FUNCTION_BLOCK FB_PrintModule_WEU_View
VAR
  // helper
  bInit   : BOOL;
  
  // config
  _pModule : POINTER TO FB_PrintModule_WEU;
  _pPositioning : POINTER TO FB_PrintPositionDmax;
  
  fbCTTrackerView : FB_CTTrackerView;
  
  // view selections
  nSelWorkerPrint : UDINT := 1;
  bShowFineAlignement : BOOL;
  // hardware view
  bShowPhDetail : BOOL;
  nSelPhDetail : UDINT := 1;
  bShowPcDetail : BOOL;
  nSelPcDetail : UDINT := 1;
  
  // motion and position view
  bShowPositionDetail : BOOL;
  bMovingInd : BOOL;
  fSpeed  : LREAL;
  fbBlink_Moving : FB_BLINK;
  
  // debug view
  bShowDebugAndSim : BOOL;
  
  fbBlink_Printing : FB_BLINK;
  bBlinkPrint : BOOL;
  bPrintInd : ARRAY[1..GVL_WEU.nC_MaxWorkerPrintPerPm] OF BOOL;
  fMaxPos : LREAL;
  t : TIME;
  zPos_PM : UDINT;
  i : UDINT;
END_VAR

VAR CONSTANT
  nC_MAX_WORKER_VIEWS : UINT := 10;
END_VAR

IF NOT checkConfig() THEN RETURN; END_IF    // check config

// -- show moving -----------------------
fSpeed := _pPositioning^.getSpeed();
IF LrealIsNaN(x:=fSpeed) THEN
  fSpeed := 0;
END_IF
t := LREAL_TO_TIME(1000-fSpeed*900);
fbBlink_Moving(bI_Enable:=SEL(fSpeed > 0, FALSE, TRUE), tI_Time:=t, bO_Out=>bMovingInd);

t := T#400MS;
fbBlink_Moving(bI_Enable:=TRUE, tI_Time:=t, bO_Out=>bBlinkPrint);
FOR i:=1 TO GVL_WEU.nC_MaxWorkerPrintPerPm DO
  bPrintInd[i] := _pModule^.fbWorkerPrint[i].bPrinting AND bBlinkPrint;
  fMaxPos := MAX(_pModule^.fbWorkerPrint[i].fPosition, fMaxPos);
END_FOR


// -- show pm module position
zPos_PM := SEL(_pModule^._pModuleMachineState^.bUnitInPrintPosition, 0, 40);

// -- show pg in p,
nSelWorkerPrint := LIMIT(1, nSelWorkerPrint, GVL_WEU.nC_MaxWorkerPrintPerPm);

// -- show ph detail
nSelPhDetail := LIMIT(1, nSelPhDetail, _pModule^._nPh);
nSelPcDetail := LIMIT(1, nSelPcDetail, _pModule^._nPc);

// -- CTTracker overview view
fbCTTrackerView.fX_m  := fMaxPos + 0.1;
fbCTTrackerView.fY_m  := 1;
fbCTTrackerView.nX_px := 300;
fbCTTrackerView.nY_px := 100;
fbCTTrackerView.fPxToMRatio := fbCTTrackerView.nX_px / fbCTTrackerView.fX_m;
fbCTTrackerView.iPrintPosition :=_pPositioning^;
fbCTTrackerView();

METHOD checkConfig : BOOL
VAR_INPUT
END_VAR
VAR_INST
  _fX_m, _fY_m   : LREAL;
  _nX_px, _nY_px : DINT; 
END_VAR
VAR
  bOK : BOOL;
END_VAR
IF NOT bInit THEN RETURN; END_IF

checkConfig := TRUE;
END_METHOD

METHOD init : BOOL
VAR_INPUT
  pModule : POINTER TO FB_PrintModule_WEU;
  pPositioning : POINTER TO FB_PrintPositionDmax;
END_VAR
IF pPositioning = 0 OR pModule = 0 THEN RETURN; END_IF

_pModule := pModule;
_pPositioning := pPositioning;

// cttracker overview
fbCTTrackerView.init(pCTTracker:=ADR(_pModule^.fbCTTracker));

bInit := TRUE;
END_METHOD

END_FUNCTION_BLOCK

(* stored: Version 1.1.0.1, ProductVersion 3.1.4024.11
   POU FB_PrintModule_WEU_View: Id {0c60165d-b9fe-4197-abbc-021f54fc96e3}, SpecialFunc None
   Method checkConfig: Id {b3643482-30cc-4825-8bf2-b809ea93dbc5}
   Method init: Id {9d295307-4d42-4a9e-9c3e-63380e114cc9} *)
